FUNCTION_BLOCK FINAL FB_MoveC EXTENDS FB_StatusExecuteFB IMPLEMENTS ITF_ExtendsFB
VAR_IN_OUT
	fbMover								: MC_PlanarMover;
END_VAR
VAR_INPUT
	Execute								: BOOL;
	Position							: DUT_Position;
	Velocity							: LREAL;
	Acceleration						: LREAL;
	Deceleration						: LREAL;
	Jerk								: LREAL;
END_VAR
VAR_OUTPUT
	Done								: BOOL;
	Busy								: BOOL;
	CommandAborted						: BOOL;
	Error								: BOOL;
	ErrorID								: UDINT;
END_VAR
VAR
	uiState								: UINT;
	//Input 内部変数
	xycPosition							: PositionXYC;
	dutPosition							: DUT_Position;
	lrVelocity							: LREAL;
	lrAcceleration						: LREAL;
	lrDeceleration						: LREAL;
	lrJerk								: LREAL;
	
	//ローカル
	fbFB_Mover							: MC_PlanarFeedback;
	fbConstraint						: DynamicConstraint_PathXY;
	stMoveCOptions						: ST_MoveCOptions;
END_VAR

Prop_Execute := Execute;
METH_Main();

fbFB_Mover.Update();

Busy := bBusy;
Done := bDone;
CommandAborted := bCommandAborted;
Error := bError;
ErrorID := udiErrorID;

//{error 'add method implementation or delete method to use base implementation'}
METHOD METH_Busy : BOOL
IF fbFB_Mover.Error THEN
	METH_Error();
	Prop_ErrorID := fbFB_Mover.ErrorId; //Moverがエラー
	RETURN;
END_IF
IF THIS^.fbMover.MCTOPLC.STD.State = MC_PLANAR_STATE.Error THEN
	METH_Error();
	Prop_ErrorID := 1; //Moverがエラー
	RETURN;
END_IF
IF fbFB_Mover.Aborted THEN
	METH_CommandAborted();
	RETURN;
END_IF

CASE THIS^.uiState OF
	0:
	fbConstraint.SetValuesVADJ(V:= THIS^.lrVelocity, A:= THIS^.lrAcceleration, D:= THIS^.lrDeceleration, J:= THIS^.lrJerk);
	//ノンモジュロ設定有効
	stMoveCOptions.direction := Tc3_Mc3PlanarMotion.MC_DIRECTION.mcDirectionNonModulo;
	THIS^.fbMover.MoveC(
		commandFeedback:= fbFB_Mover, 
		targetPosition:= dutPosition.c, 
		constraint:= fbConstraint, 
		options:= stMoveCOptions);
	THIS^.uiState := 10;	
	
	10:
	IF fbFB_Mover.Done THEN
		THIS^.uiState := 16#FFFF;	
	END_IF
	
	16#FFFF:
	METH_Done();
END_CASE
END_METHOD

//{error 'add method implementation or delete method to use base implementation'}
METHOD METH_Enter : BOOL
//Input 内部変数に移す
dutPosition := Position;
lrVelocity := Velocity;
lrAcceleration := Acceleration;
lrDeceleration := Deceleration;
lrJerk := Jerk;
END_METHOD

//{error 'add method implementation or delete method to use base implementation'}
METHOD METH_Exit : BOOL
Prop_Done := FALSE;
Prop_Busy := FALSE;
Prop_CommandAborted := FALSE;
Prop_Error := FALSE;
Prop_ErrorID := 0;

// 内部変数をリフレッシュする
uiState := 0;
xycPosition.SetValuesXYC(0,0,0);
lrVelocity := 0;
lrAcceleration := 0;
lrDeceleration := 0;
lrJerk := 0;
END_METHOD

//{error 'add method implementation or delete method to use base implementation'}
METHOD METH_Main : BOOL
//Doneに遷移
IF SUPER^.bDone AND SUPER^.bExecute THEN
	METH_Done();
	RETURN;
END_IF
//Errorに遷移
IF SUPER^.bError AND SUPER^.bExecute THEN
	METH_Error();
	RETURN;
END_IF
//CommandAbortedに遷移
IF SUPER^.bCommandAborted AND SUPER^.bExecute THEN
	METH_CommandAborted();
	RETURN;
END_IF
//FBをリフレッシュ
//状態がDone, Error, CommandAborted時に Execute FALSE で遷移
IF (SUPER^.bDone OR SUPER^.bError OR SUPER^.bCommandAborted) AND NOT SUPER^.bExecute THEN
	METH_Exit();
	RETURN;
END_IF

//実行開始
IF SUPER^.bExecute AND NOT SUPER^.bBusy THEN
	METH_Execute();
	METH_Enter();
END_IF
//実行中
IF SUPER^.bBusy THEN
	METH_Busy();
END_IF
END_METHOD

END_FUNCTION_BLOCK

(* stored: Version 1.1.0.1, ProductVersion 3.1.4024.11
   POU FB_MoveC: Id {2a4ddaa4-4554-4520-af71-d3cc30323ba1}, SpecialFunc None
   Method METH_Busy: Id {4b15cace-e6e9-4756-8aee-363e63ee931d}
   Method METH_Enter: Id {b4ad9405-bcca-40f1-8d0f-a7ff72000c1b}
   Method METH_Exit: Id {792bcaaf-1c95-49d6-85d3-214c2cec9094}
   Method METH_Main: Id {985bdbbf-de12-429c-9993-2e6090ee64c5} *)
